TYPE ST_HW_OutputsClosedPalletCheck :
STRUCT		

END_STRUCT
END_TYPE

(* stored: Version 1.1.0.1, ProductVersion 3.1.4024.9
   DUT ST_HW_OutputsClosedPalletCheck: Id {2e620b87-0612-48d4-a9ee-654aae57d22a} *)
